// TIA Portal V19 export
FUNCTION "SERVICE PRODUCTION" : Void   // FC20, STL
TITLE = CASCADE REGULATOR FOR TT55.62 / TT55.60
{ S7_Optimized_Access := 'TRUE' }
NAME : PRODSERV
VERSION : 0.0
// Programmer Init: 8242-BUG
// 
// Change Log:
// 
// Date        Change                          Updated by
// ------------------------------------------------------
// 12.09.00    1. Edition                      BUG
// 17.07.01    2. Edition                      BUG
//                - temp offset
// stored: AutoNumber false
   VAR_TEMP
      __PlcmigTempFillBits_0B0 : Array[0..7] of Bool;
   END_VAR
BEGIN

NETWORK
TITLE = Q 28.1; Output modul 3 Channel 1
// Cascade regulator Auto/Man/off
      A     "B01.65";
      O     "HSL0165_Proxy";  // it manuel, cascade not controlling

      =     "M_AHV_HIGH_LEVEL";
      A     "TANK STERILE";  // if auto, cascade is controlling

      =     "M_AHV_STERILE";
      AN    "MY0101";  // add offset when steril
      A     "Y0101R";
      =     "M_AHV_CLOSED";
      A     "DUMMY PROD. AT FILLING";  // if off, setpoint = PID setpoint

      A     "TANK STERILE";
      =     "M_PROD_AVAILABLE";  // add offset when controller is off
      AN    "S0 PRODUCTION TANK";
      R     "FILLING PIPE DRAINED";
      R     "DUMMY1 DRAIN";  // if off, setpoint = PID setpoint

      R     "DUMMY2 DRAIN";
      JC    M001;
      L     "Setpoints".PT0167SpProduction;
      T     "STP_PT0167/IP0149_50".PT0167SpSTP;
      A     "FILLING PIPE DRAINED";
      JC    M001;
      A     "DUMMY2 DRAIN";
      JC    M002;
      A     "DUMMY1 DRAIN";
      JC    M003;
      A     "MY0101";
      JC    M004;
      JU    M001;
M002: A     "T 45 PURGE";
      JC    M001;
      R     "MY0112";
      R     "MY0113";
      S     "FILLING PIPE DRAINED";
      R     "DUMMY2 DRAIN";
      JU    M001;
M003: A     "T 44 FILLING DRAIN";
      JC    M001;
      S     "MY0112";
      S     "MY0113";
      S     "MY0114";
      S     "DUMMY2 DRAIN";
      S     "TIM45";
      R     "DUMMY1 DRAIN";
      JU    M001;
M004: S     "TIM44";
      AN    "GS22_62";
      AN    "GS22_68";
      A     "GS22_61";
      A     "GS22_63";
      S     "DUMMY1 DRAIN";
      A     "GS22_62";
      A     "GS22_68";
      AN    "GS22_61";
      AN    "GS22_63";
      S     "FILLING PIPE DRAINED";
M001: NOP   0;

NETWORK
TITLE = DUMMY PRODUCT AT FILLING MASHINES
// Load TT5560 - Delta, to setpoint when sterile product at A-Tank
      AN    "TANK STERILE";
      JC    M005;  // dummy
      AN    "B01.66";

      JC    M005;
      AN    "FILLING PIPE DRAINED";
      JC    M005;
      A     "DUMMY PROD. AT FILLING";
      JC    M006;
      S     "DUMMY PROD. AT FILLING";
      S     "ProcessAndPbAlarms"."A"[52];  //A52_ProdAtFillingMash
      JU    M006;
M005: R     "DUMMY PROD. AT FILLING";
M006: NOP   0;

NETWORK
TITLE = A49_TankFull
// Cascade regulator Auto
// WAIT UNTIL TIMER EXPIRES THEN TEST AND CALCULATE AGAIN
      CLR;  // 60 SEC DELAY
      A     "StopFillers_UHT_Rec";
      JC    M007;
      AN    "S0 PRODUCTION TANK";
      JC    M007;
      AN    "TANK STERILE";
      JC    M007;  // 60 SEC DELAY
      A     "B01.65";
      O     "HSL0165_Proxy";
      S     "ProcessAndPbAlarms"."A"[49];  //A49_TankFull
      JC    M007;
      S     "M_AHV_READY";
      S     "S.T.01.TANK READY";
      JU    M008;
M007: NOP   0;
      R     "M_AHV_READY";
      R     "S.T.01.TANK READY";
M008: NOP   0;

NETWORK
TITLE = AGITATOR IN AUTOMATIC MODE
// TEST IF MEASURED VALUE IS WITHIN LIMITS
      A     "S0 PRODUCTION TANK";
      A     "FILLING PIPE DRAINED";
      AN    "B01.66";
      R     "AGITATOR AUTOMATIC";
      =     "ProcessAndPbAlarms"."A"[48];  //A48_TankEmpty

NETWORK
TITLE = 
      AN    "FLIP 01.44";
      JC    M009;
      A     "T 52 FLIP 01.44";
      JC    M009;
      A     "MY0144";
      JC    M00a;
      S     "MY0144";
      S     "TIM52";
      JU    M009;
M00a: R     "MY0144";
      R     "FLIP 01.44";
M009: NOP   0;

NETWORK
TITLE = 
      A     "TANK AUTO";
      AN    "Tag_56";
      S     "Tag_57";

NETWORK
TITLE = 
      A     "TANK AUTO";
      A     "Tag_57";
      L     S5T#6M;
      SD    "Tag_56";
      NOP   0;
      NOP   0;
      NOP   0;
      A     "Tag_56";
      =     #__PlcmigTempFillBits_0B0[0];
      A     #__PlcmigTempFillBits_0B0[0];
      JNB   M00b;
      L     "OP25 TANK".RuninghoursAHV;
      L     0.1;
      +R;
      T     "OP25 TANK".RuninghoursAHV;
M00b: NOP   0;
      A     #__PlcmigTempFillBits_0B0[0];
      BLD   102;
      R     "Tag_57";

NETWORK
TITLE = 
      A     "LEDAssignment".ResetTotaliserHoursAHV;
      =     #__PlcmigTempFillBits_0B0[0];
      A     #__PlcmigTempFillBits_0B0[0];
      JNB   M00c;
      L     0.0;
      T     "OP25 TANK".RuninghoursAHV;
M00c: NOP   0;
      A     #__PlcmigTempFillBits_0B0[0];
      BLD   102;
      R     "LEDAssignment".ResetTotaliserHoursAHV;

NETWORK
TITLE = 
      O     "Set_alarm_lamp_feedback";
      O     "Set_alarm_lamp_monitor";
      O     "Set_alarm_lamp_process";
      =     "S.T.01.NOT USED 8";
END_FUNCTION
